screen "83_КалібровкаКрану" 800x454, template "Template_1"
   on GenerateScreen: SetTag("Tag_ScreenNumber", 83)
   IOField "I/O field_3" at 365,32 size 70x25; FormatPattern 99999
      ProcessValue <- "HMI_DB_Calibration_Crane_CurrentStep"
   IOField "I/O field_4" at 365,32 size 70x25; FormatPattern 99999
      ProcessValue <- "HMI_DB_Calibration_Crane_CurrentStep"
      Visibility <- "HMI_DB_Calibration_Crane_Calibrated"
   IOField "I/O field_5" at 365,32 size 70x25; FormatPattern 99999
      ProcessValue <- "HMI_DB_Calibration_Crane_CurrentStep"
      Visibility <- "HMI_DB_Calibration_Crane_Active"
   IOField "I/O field_6" at 365,32 size 70x25; FormatPattern 99999
      ProcessValue <- "HMI_DB_Calibration_Crane_CurrentStep"
      Visibility <- "HMI_DB_Calibration_Crane_Aborted"
   IOField "I/O field_7" at 365,32 size 70x25; FormatPattern 99999
      ProcessValue <- "HMI_DB_Calibration_Crane_CurrentStep"
      Visibility <- "HMI_DB_Calibration_Crane_Fault"
   TextField "Text field_12" at 681,263 size 30x18; Text '110'
   TextField "Text field_13" at 23,263 size 22x18; Text '10'
   TextField "Text field_14" at 89,263 size 22x18; Text '20'
   TextField "Text field_15" at 155,263 size 22x18; Text '30'
   TextField "Text field_16" at 221,263 size 22x18; Text '40'
   TextField "Text field_17" at 288,263 size 22x18; Text '50'
   TextField "Text field_18" at 354,263 size 22x18; Text '60'
   TextField "Text field_19" at 420,263 size 22x18; Text '70'
   TextField "Text field_20" at 486,263 size 22x18; Text '80'
   TextField "Text field_21" at 553,263 size 22x18; Text '90'
   TextField "Text field_22" at 615,263 size 30x18; Text '100'
   TextField "Text field_24" at 748,263 size 30x18; Text '130'
   TextField "Text field_5" at 8,101 size 61x18; Text 'Позиція'
   TextField "Text field_6" at 8,166 size 136x18; Text 'Реперний вимикач'
   TextField "Text field_7" at 8,121 size 80x18; Text 'Швидкість'
   TextField "Text field_8" at 365,142 size 104x18; Text 'Залишок часу'
   IOField "I/O field_1" at 136,98 size 120x25; FormatPattern s999999
      ProcessValue <- "HMI_DB_Calibration_Crane_Position4BR1_mm"
   IOField "I/O field_2" at 136,118 size 120x25; FormatPattern s9999.99
      ProcessValue <- "HMI_DB_Calibration_Crane_Drive1Velocity_rpm"
   Circle "Circle_49" at 211,167 size 16x16
      Appearance <- "HMI_DB_Calibration_Crane_Reference4K1"
   TextField "Text field_9" at 47,5 size 247x21; Text 'Статус калібровки мех. крану'
   TextField "Text field_10" at 482,5 size 181x21; Text 'Поточний крок та дія'
   Group "Group_1" at 365,32 size 70x25
   SymbolicIOField "Symbolic I/O field_1" at 453,29 size 327x32; TextOff '0'; TextOn '1'; TextList "CraneStepName"
      ProcessValue <- "HMI_DB_Calibration_Crane_CurrentStep"
   TextField "Text field_11" at 365,102 size 268x18; Text 'Умови переходу на наступний крок:'
   SymbolicIOField "Symbolic I/O field_2" at 365,115 size 416x32; TextOff '0'; TextOn '1'; TextList "CraneCondition"
      ProcessValue <- "HMI_DB_Calibration_Crane_CurrentStep"
   Group "Group_2" at 680,256 size 32x32
   Group "Group_3" at 18,256 size 32x32
   Group "Group_4" at 84,256 size 32x32
   Group "Group_5" at 150,256 size 32x32
   Group "Group_6" at 216,256 size 32x32
   Group "Group_7" at 283,256 size 32x32
   Group "Group_8" at 349,256 size 32x32
   Group "Group_9" at 415,256 size 32x32
   Group "Group_10" at 481,256 size 32x32
   Group "Group_11" at 548,256 size 32x32
   Group "Group_12" at 614,256 size 32x32
   Group "Group_14" at 747,256 size 32x32
   TextField "Text field_23" at 0,295 size 68x28; Text 'Перевірка умов'
   TextField "Text field_25" at 68,295 size 65x40; Text 'Натисніть кнопку "Вліво"'
   TextField "Text field_26" at 133,295 size 67x40; Text 'Рух до реперної точки 4К1'
   TextField "Text field_27" at 198,295 size 69x40; Text 'Відпустіть кнопку "Вліво"'
   TextField "Text field_28" at 263,295 size 85x40; Text 'Перемістить механізм від 4К1'
   TextField "Text field_29" at 330,295 size 70x28; Text 'Відхід завершено'
   TextField "Text field_30" at 399,295 size 65x40; Text 'Натисніть кнопку "Вліво"'
   TextField "Text field_31" at 462,295 size 70x40; Text 'Повторний підхід до 4К1'
   TextField "Text field_32" at 544,295 size 40x28; Text 'Quick Stop'
   TextField "Text field_33" at 593,295 size 75x40; Text 'Очікування зупинки приводів'
   TextField "Text field_34" at 665,295 size 66x40; Text 'Запуск preset енкодерів'
   TextField "Text field_35" at 725,295 size 75x40; Text 'Калібровку успішно завершено'
   Group "Group_13" at 26,342 size 16x16
   Group "Group_15" at 92,342 size 16x16
   Group "Group_16" at 158,342 size 16x16
   Group "Group_17" at 224,342 size 16x16
   Group "Group_18" at 291,342 size 16x16
   Group "Group_19" at 357,342 size 16x16
   Group "Group_20" at 423,342 size 16x16
   Group "Group_21" at 489,342 size 16x16
   Group "Group_22" at 556,342 size 16x16
   Group "Group_23" at 622,342 size 16x16
   Group "Group_24" at 688,342 size 16x16
   Group "Group_25" at 755,342 size 16x16
   TextField "Text field_36" at 18,381 size 148x18; Text 'Умовні позначення:'
   TextField "Text field_37" at 190,381 size 85x18; Text '- Виконано'
   TextField "Text field_38" at 365,381 size 124x18; Text '- Поточний крок'
   TextField "Text field_39" at 540,381 size 92x18; Text '- Очікується'
   TextField "Text field_40" at 218,226 size 367x21; Text 'Послідовність кроків калібровки мех. крану'
   IOField "I/O field_8" at 540,139 size 60x25; FormatPattern 999; Unit  хв :
      ProcessValue <- "HMI_DB_Calibration_Crane_TimerRemaining_Min"
   IOField "I/O field_9" at 594,139 size 55x25; FormatPattern 999; Unit  сек
      ProcessValue <- "HMI_DB_Calibration_Crane_TimerRemaining_Sec"
   TextField "Text field_42" at 8,141 size 88x18; Text 'Інкременти'
   IOField "I/O field_10" at 136,138 size 80x25; FormatPattern s99999999
      ProcessValue <- "RawPosition"
   Group "Group" at 38,33 size 258x23
   TextField "Text field_43" at 8,191 size 220x18; Text 'Дозв. від мех. підйому і візка'
   Circle "Circle_53" at 211,192 size 16x16
      Appearance <- "HMI_DB_Calibration_Crane_PrerequisitesNotOK"
   IOField "I/O field_11" at 224,98 size 120x25; FormatPattern s999999; Unit  мм
      ProcessValue <- "HMI_DB_Calibration_Crane_Position4BR2_mm"
   IOField "I/O field_12" at 224,118 size 120x25; FormatPattern s9999.99; Unit  об/хв
      ProcessValue <- "HMI_DB_Calibration_Crane_Drive2Velocity_rpm"
   IOField "I/O field_13" at 227,138 size 80x25; FormatPattern s99999999
      ProcessValue <- "RawPosition"
   Circle "Circle_14" at 26,342 size 16x16
      Visibility <- "HMI_DB_Calibration_Crane_Steps_Active_Step10"
   Circle "Circle_15" at 26,342 size 16x16
      Visibility <- "HMI_DB_Calibration_Crane_Steps_Completed_Step10"
   Circle "Circle_17" at 92,342 size 16x16
      Visibility <- "HMI_DB_Calibration_Crane_Steps_Active_Step20"
   Circle "Circle_18" at 92,342 size 16x16
      Visibility <- "HMI_DB_Calibration_Crane_Steps_Completed_Step20"
   Circle "Circle_20" at 158,342 size 16x16
      Visibility <- "HMI_DB_Calibration_Crane_Steps_Active_Step30"
   Circle "Circle_21" at 158,342 size 16x16
      Visibility <- "HMI_DB_Calibration_Crane_Steps_Completed_Step30"
   Circle "Circle_23" at 224,342 size 16x16
      Visibility <- "HMI_DB_Calibration_Crane_Steps_Active_Step40"
   Circle "Circle_24" at 224,342 size 16x16
      Visibility <- "HMI_DB_Calibration_Crane_Steps_Completed_Step40"
   Circle "Circle_26" at 291,342 size 16x16
      Visibility <- "HMI_DB_Calibration_Crane_Steps_Active_Step50"
   Circle "Circle_27" at 291,342 size 16x16
      Visibility <- "HMI_DB_Calibration_Crane_Steps_Completed_Step50"
   Circle "Circle_29" at 357,342 size 16x16
      Visibility <- "HMI_DB_Calibration_Crane_Steps_Active_Step60"
   Circle "Circle_30" at 357,342 size 16x16
      Visibility <- "HMI_DB_Calibration_Crane_Steps_Completed_Step60"
   Circle "Circle_32" at 423,342 size 16x16
      Visibility <- "HMI_DB_Calibration_Crane_Steps_Active_Step70"
   Circle "Circle_33" at 423,342 size 16x16
      Visibility <- "HMI_DB_Calibration_Crane_Steps_Completed_Step70"
   Circle "Circle_35" at 489,342 size 16x16
      Visibility <- "HMI_DB_Calibration_Crane_Steps_Active_Step80"
   Circle "Circle_36" at 489,342 size 16x16
      Visibility <- "HMI_DB_Calibration_Crane_Steps_Completed_Step80"
   Circle "Circle_38" at 556,342 size 16x16
      Visibility <- "HMI_DB_Calibration_Crane_Steps_Active_Step90"
   Circle "Circle_39" at 556,342 size 16x16
      Visibility <- "HMI_DB_Calibration_Crane_Steps_Completed_Step90"
   Circle "Circle_41" at 622,342 size 16x16
      Visibility <- "HMI_DB_Calibration_Crane_Steps_Active_Step100"
   Circle "Circle_42" at 622,342 size 16x16
      Visibility <- "HMI_DB_Calibration_Crane_Steps_Completed_Step100"
   Circle "Circle_44" at 688,342 size 16x16
      Visibility <- "HMI_DB_Calibration_Crane_Steps_Active_Step110"
   Circle "Circle_45" at 688,342 size 16x16
      Visibility <- "HMI_DB_Calibration_Crane_Steps_Completed_Step110"
   Circle "Circle_47" at 755,342 size 16x16
      Visibility <- "HMI_DB_Calibration_Crane_Steps_Active_Step130"
   Circle "Circle_48" at 755,342 size 16x16
      Visibility <- "HMI_DB_Calibration_Crane_Steps_Completed_Step130"
   TextField "Text field_41" at 83,33 size 169x23; Text 'НЕ КАЛІБРОВАНО'
      Visibility <- "HMI_DB_Calibration_Crane_Calibrated"
   TextField "Text field_4" at 38,33 size 258x23; Text 'КАЛІБРОВКА АНУЛЬОВАНА'
      Visibility <- "HMI_DB_Calibration_Crane_Aborted"
   TextField "Text field_2" at 58,33 size 219x23; Text 'КАЛІБРОВКА АКТИВНА'
      Visibility <- "HMI_DB_Calibration_Crane_Active"
   TextField "Text field_3" at 56,33 size 223x23; Text 'ПОМИЛКА КАЛІБРОВКИ'
      Visibility <- "HMI_DB_Calibration_Crane_Fault"
   TextField "Text field_1" at 98,33 size 139x23; Text 'КАЛІБРОВАНО'
      Visibility <- "HMI_DB_Calibration_Crane_Calibrated"
   TextField "Text field_44" at 149,77 size 75x18; Text '4М1'
   TextField "Text field_45" at 221,77 size 75x18; Text '4М2'
   Group "Group_26" at 207,61 size 25x0
   Line "Line_4" at 207,61 size 25x0
      Visibility <- "HMI_DB_Crane_movement_mechanism_FirstSpeedRight"
   Line "Line_5" at 207,61 size 25x0
      Visibility <- "HMI_DB_Crane_movement_mechanism_FirstSpeedLeft"

screen "70_Діагностика" 800x454, template "Template_1"
   on GenerateScreen: SetTag("Tag_ScreenNumber", 70); function_c655a98f("HMI_Connection_1", "HMI_PLC_Mode"); "HMI_UpdateCommunication"()
   TextField "Text field_1" at 166,42 size 46x23; Text 'A1.1'
   TextField "Text field_2" at 166,216 size 46x23; Text 'A1.0'
   TextField "Text field_3" at 715,26 size 41x23; Text '1BR'
   TextField "Text field_4" at 715,115 size 41x23; Text '3BR'
   TextField "Text field_5" at 710,206 size 52x23; Text '4BR1'
   TextField "Text field_6" at 710,295 size 52x23; Text '4BR2'
   TextField "Text field_7" at 436,67 size 46x23; Text 'A1.6'
   TextField "Text field_8" at 348,286 size 23x18; Text 'U1'
   TextField "Text field_9" at 394,286 size 40x18; Text '1UZ1'
   TextField "Text field_10" at 436,286 size 40x18; Text '3UZ1'
   TextField "Text field_11" at 479,286 size 40x18; Text '4UZ1'
   TextField "Text field_12" at 522,286 size 40x18; Text '4UZ2'
   Button "Button_3" at 4,10 size 104x34; TextOff 'Діагностика / Тренди'; TextOn 'Діагностика'
      on Release: ActivateScreen("50_Trends(1UZ1)", 0)
   TextField "PN_Status_DisplayOpen" at 120,1 size 550x20; Text 'MRP: RING OPEN / MRP: КІЛЬЦЕ РОЗІМКНЕНЕ'
      Visibility <- "HMI_Show_RingOpen"
   TextField "PN_Status_DisplayClosed" at 120,0 size 550x20; Text 'MRP: RING CLOSED / MRP: КІЛЬЦЕ ЗАМКНЕНЕ'
      Visibility <- "HMI_Show_RingClosed"
   TextField "PN_Status_DisplayUnknown" at 120,20 size 550x20; Text 'PN: DIAGNOSTIC DATA UNAVAILABLE / PN: ДІАГНОСТИЧНІ ДАНІ НЕДОСТУПНІ'
      Visibility <- "HMI_Show_DiagnosticsUnknown"
   TextField "PN_Status_DisplayHmiFault" at 120,20 size 550x20; Text 'HMI: PLC DETECTED A PANEL COMMUNICATION FAULT / HMI: ПЛК ВИЯВИВ ПОРУШЕННЯ ОБМІНУ З ПАНЕЛЛЮ'
      Visibility <- "HMI_Show_PanelFault"
   TextField "HMI_Status_NoConnection" at 120,20 size 550x20; Text 'HMI: NO COMMUNICATION BETWEEN PLC AND OPERATOR PANEL / HMI: НЕМАЄ ЗВʼЯЗКУ МІЖ ПЛК І ПАНЕЛЛЮ ОПЕРАТОРА'
      Visibility <- "HMI_Show_NoConnection"
   TextField "HMI_Status_CpuStopped" at 120,20 size 550x20; Text 'PLC: STOPPED. DIAGNOSTICS ARE NOT UPDATING / ПЛК: ЗУПИНЕНО (STOP). ДІАГНОСТИКА НЕ ОНОВЛЮЄТЬСЯ'
      Visibility <- "HMI_Show_CpuStopped"
   TextField "HMI_Status_CpuUnknown" at 120,20 size 550x20; Text 'PLC: RUN MODE NOT CONFIRMED / ПЛК: РЕЖИМ RUN НЕ ПІДТВЕРДЖЕНО'
      Visibility <- "HMI_Show_CpuUnknown"
   GraphicView "Graphic view_1" at 64,63 size 255x119; Picture "plc"
   GraphicView "Graphic view_2" at 428,91 size 62x124; Picture "scalance"
   GraphicView "Graphic view_3" at 697,30 size 76x48; Picture "6FX2001-5QN25_P_NC01_XX_01618I"
   GraphicView "Graphic view_5" at 343,307 size 46x80; Picture "6SL3040-1MA01-0AA0_P_D211_XX_00205P"
   GraphicView "Graphic view_6" at 697,119 size 76x48; Picture "6FX2001-5QN25_P_NC01_XX_01618I"
   GraphicView "Graphic view_7" at 697,209 size 76x48; Picture "6FX2001-5QN25_P_NC01_XX_01618I"
   GraphicView "Graphic view_8" at 697,299 size 76x48; Picture "6FX2001-5QN25_P_NC01_XX_01618I"
   GraphicView "Graphic view_4" at 100,239 size 184x118; Picture "hmi_1"
   GraphicView "Graphic view_9" at 389,301 size 50x90; Picture "6SL3210-1PE14-3UL1_P_D011_XX_00576_4_1"
   GraphicView "Graphic view_10" at 431,301 size 50x90; Picture "6SL3210-1PE14-3UL1_P_D011_XX_00576_4_1"
   GraphicView "Graphic view_11" at 474,301 size 50x90; Picture "6SL3210-1PE14-3UL1_P_D011_XX_00576_4_1"
   GraphicView "Graphic view_12" at 517,301 size 50x90; Picture "6SL3210-1PE14-3UL1_P_D011_XX_00576_4_1"
   Group "NOK_A1.5" at 276,66 size 40x111
   Group "NOK_A1.4" at 233,66 size 40x111
   Group "NOK_A1.3" at 192,66 size 40x111
   Group "NOK_A1.2" at 147,66 size 40x111
   Group "NOK_A1.1" at 66,66 size 77x111
   GraphicView "Graphic view_21" at 343,309 size 45x80; Picture "Graphic_4"
      Visibility <- "HMI_DB_Alarms_Diagn_AlarmWord1"
   GraphicView "Graphic view_20" at 391,309 size 45x80; Picture "Graphic_4"
      Visibility <- "HMI_DB_Alarms_Diagn_AlarmWord1"
   GraphicView "Graphic view_19" at 431,309 size 45x80; Picture "Graphic_4"
      Visibility <- "HMI_DB_Alarms_Diagn_AlarmWord1"
   GraphicView "Graphic view_18" at 479,309 size 45x80; Picture "Graphic_4"
      Visibility <- "HMI_DB_Alarms_Diagn_AlarmWord1"
   GraphicView "Graphic view_17" at 519,309 size 45x80; Picture "Graphic_4"
      Visibility <- "HMI_DB_Alarms_Diagn_AlarmWord1"
   GraphicView "Graphic view_16" at 688,290 size 85x80; Picture "Graphic_4"
      Visibility <- "HMI_DB_Alarms_Diagn_AlarmWord1"
   GraphicView "Graphic view_15" at 688,202 size 85x80; Picture "Graphic_4"
      Visibility <- "HMI_DB_Alarms_Diagn_AlarmWord1"
   GraphicView "Graphic view_14" at 688,114 size 85x80; Picture "Graphic_4"
      Visibility <- "HMI_DB_Alarms_Diagn_AlarmWord1"
   GraphicView "Graphic view_13" at 688,26 size 85x80; Picture "Graphic_4"
      Visibility <- "HMI_DB_Alarms_Diagn_AlarmWord1"
   GraphicView "Graphic view_22" at 416,96 size 85x106; Picture "Graphic_4"
      Visibility <- "HMI_DB_Alarms_Diagn_AlarmWord1"
   GraphicView "Graphic view_23" at 279,348 size 40x70; Picture "Graphic_4"
      Visibility <- "HMI_Show_Cross_HMI_CU"
   GraphicView "Graphic view_24" at 287,172 size 40x70; Picture "Graphic_4"
      Visibility <- "HMI_Show_Cross_PLC_SC"
   GraphicView "Graphic view_25" at 112,348 size 40x70; Picture "Graphic_4"
      Visibility <- "HMI_Show_Cross_PLC_HMI"
   GraphicView "Graphic view_26" at 383,204 size 40x70; Picture "Graphic_4"
      Visibility <- "HMI_Show_Cross_SC_CU"
   Line "Line_8" at 276,66 size 40x111
      Visibility <- "HMI_DB_Alarms_Diagn_AlarmWord1"
   Line "Line_9" at 276,66 size 40x111
      Visibility <- "HMI_DB_Alarms_Diagn_AlarmWord1"
   Line "Line_1" at 233,66 size 40x111
      Visibility <- "HMI_DB_Alarms_Diagn_AlarmWord1"
   Line "Line_2" at 233,66 size 40x111
      Visibility <- "HMI_DB_Alarms_Diagn_AlarmWord1"
   Line "Line_3" at 192,66 size 40x111
      Visibility <- "HMI_DB_Alarms_Diagn_AlarmWord1"
   Line "Line_4" at 192,66 size 40x111
      Visibility <- "HMI_DB_Alarms_Diagn_AlarmWord1"
   Line "Line_5" at 147,66 size 40x111
      Visibility <- "HMI_DB_Alarms_Diagn_AlarmWord1"
   Line "Line_6" at 147,66 size 40x111
      Visibility <- "HMI_DB_Alarms_Diagn_AlarmWord1"
   Line "Line_7" at 66,66 size 77x111
      Visibility <- "HMI_DB_Alarms_Diagn_AlarmWord1"
   Line "Line_10" at 66,66 size 77x111
      Visibility <- "HMI_DB_Alarms_Diagn_AlarmWord1"
   Button "btn1BR" at 690,32 size 90x45; TextOff 'Text'
      on Release: ActivateScreen("77_1BR", 0)
   Button "btn3BR" at 690,121 size 90x45; TextOff 'Text'
      on Release: ActivateScreen("78_3BR", 0)
   Button "btn4BR1" at 690,211 size 90x45; TextOff 'Text'
      on Release: ActivateScreen("79_4BR1", 0)
   Button "btn4BR2" at 690,301 size 90x45; TextOff 'Text'
      on Release: ActivateScreen("710_4BR2", 0)
   Button "btnU1" at 330,304 size 62x92; TextOff 'Text'
      on Release: ActivateScreen("30_Drives(CU)", 0)
   Button "btnA1.2" at 147,50 size 43x119; TextOff 'Text'
      on Release: ActivateScreen("71_A1.2(DI32)_1", 0)
   Button "btnA1.3" at 189,50 size 43x119; TextOff 'Text'
      on Release: ActivateScreen("73_A1.3(DI32)_1", 0)
   Button "btnA1.4" at 233,50 size 43x119; TextOff 'Text'
      on Release: ActivateScreen("76_A1.4(IW8)", 0)
   Button "btnA1.5" at 276,50 size 43x119; TextOff 'Text'
      on Release: ActivateScreen("75_A1.5(DQ16)", 0)
   Button "btn1UZ1" at 394,304 size 35x92; TextOff 'Text'
      on Release: ActivateScreen("31_Drives(1UZ1)", 0)
   Button "btn3UZ1" at 434,304 size 37x92; TextOff 'Text'
      on Release: ActivateScreen("32_Drives(3UZ1)", 0)
   Button "btn4UZ1" at 478,304 size 37x92; TextOff 'Text'
      on Release: ActivateScreen("33_Drives(4UZ1)", 0)
   Button "btn4UZ2" at 522,304 size 37x92; TextOff 'Text'
      on Release: ActivateScreen("34_Drives(4UZ2)", 0)

VB script "StartLog"
   'Tip:
   ' 1. Use the <CTRL+SPACE> or <CTRL+I> shortcut to open a list of all objects and functions
   ' 2. Write the code using the HMI Runtime object.
   '  Example: HmiRuntime.Screens("Screen_1").
   ' 3. Use the <CTRL+J> shortcut to create an object reference.
   'Write the code as of this position:
    bb0abc73-aec8-40d0-9880-0280a6a3de42()
    fd9437ed-c09f-45a2-bbcf-d542009dcc27 $3$hmiDataLog$,1UZ1
    fd9437ed-c09f-45a2-bbcf-d542009dcc27 $3$hmiDataLog$, 3UZ1 
    fd9437ed-c09f-45a2-bbcf-d542009dcc27 $3$hmiDataLog$, 4UZ1 
    fd9437ed-c09f-45a2-bbcf-d542009dcc27 $3$hmiDataLog$,4UZ2 
    fd9437ed-c09f-45a2-bbcf-d542009dcc27 $3$hmiAlarmLog$,MessageContactor 
    fd9437ed-c09f-45a2-bbcf-d542009dcc27 $3$hmiAlarmLog$,MessageLiftUp 
    fd9437ed-c09f-45a2-bbcf-d542009dcc27 $3$hmiAlarmLog$,MessageTrolley 
    fd9437ed-c09f-45a2-bbcf-d542009dcc27 $3$hmiAlarmLog$,MessageCrane 
    fd9437ed-c09f-45a2-bbcf-d542009dcc27 $3$hmiAlarmLog$,MessageDiag 
    fd9437ed-c09f-45a2-bbcf-d542009dcc27 $3$hmiAlarmLog$,AlarmCrane 
    fd9437ed-c09f-45a2-bbcf-d542009dcc27 $3$hmiAlarmLog$,AlarmTrolley 
    fd9437ed-c09f-45a2-bbcf-d542009dcc27 $3$hmiAlarmLog$,AlarmLiftUp 
    fd9437ed-c09f-45a2-bbcf-d542009dcc27 $3$hmiAlarmLog$,AlarmContactor 
    fd9437ed-c09f-45a2-bbcf-d542009dcc27 $3$hmiAlarmLog$,AlarmDiag 
    fd9437ed-c09f-45a2-bbcf-d542009dcc27 $3$hmiAlarmLog$,MessageSelf 
    SmartTags("iStep") = 0

VB script "StopLog"
   'Tip:
   ' 1. Use the <CTRL+SPACE> or <CTRL+I> shortcut to open a list of all objects and functions
   ' 2. Write the code using the HMI Runtime object.
   '  Example: HmiRuntime.Screens "Screen_1" .
   ' 3. Use the <CTRL+J> shortcut to create an object reference.
   'Write the code as of this position:
    b6526003-1e6c-4105-b1c3-8571bad56740 $3$hmiDataLog$,1UZ1
    b6526003-1e6c-4105-b1c3-8571bad56740 $3$hmiDataLog$,3UZ1 
    b6526003-1e6c-4105-b1c3-8571bad56740 $3$hmiDataLog$,4UZ1 
    b6526003-1e6c-4105-b1c3-8571bad56740 $3$hmiDataLog$,4UZ2 
    b6526003-1e6c-4105-b1c3-8571bad56740 $3$hmiAlarmLog$,MessageContactor 
    b6526003-1e6c-4105-b1c3-8571bad56740 $3$hmiAlarmLog$,MessageLiftUp 
    b6526003-1e6c-4105-b1c3-8571bad56740 $3$hmiAlarmLog$,MessageTrolley 
    b6526003-1e6c-4105-b1c3-8571bad56740 $3$hmiAlarmLog$,MessageCrane 
    b6526003-1e6c-4105-b1c3-8571bad56740 $3$hmiAlarmLog$,MessageDiag 
    b6526003-1e6c-4105-b1c3-8571bad56740 $3$hmiAlarmLog$,AlarmCrane 
    b6526003-1e6c-4105-b1c3-8571bad56740 $3$hmiAlarmLog$,AlarmTrolley 
    b6526003-1e6c-4105-b1c3-8571bad56740 $3$hmiAlarmLog$,AlarmLiftUp 
    b6526003-1e6c-4105-b1c3-8571bad56740 $3$hmiAlarmLog$,AlarmContactor 
    b6526003-1e6c-4105-b1c3-8571bad56740 $3$hmiAlarmLog$,AlarmDiag 
    b6526003-1e6c-4105-b1c3-8571bad56740 $3$hmiAlarmLog$,MessageSelf 
    efd5fb8c-e901-419b-bc1e-08a47a763dd7  
    SmartTags("iStep")  = 1

VB script "CopyLogs"
   'Tip:
   ' 1. Use the <CTRL+SPACE> or <CTRL+I> shortcut to open a list of all objects and functions
   ' 2. Write the code using the HMI Runtime object.
   '  Example: HmiRuntime.Screens("Screen_1").
   ' 3. Use the <CTRL+J> shortcut to create an object reference.
   'Write the code as of this position:
    
    Dim st
    
    On Error Resume Next
    
    e9be9208-412d-4969-b0d9-b24c90392a10 $3$hmiDataLog$,1UZ1, "\Storage Card USB\archive\", $3$hmiCopy$
    e9be9208-412d-4969-b0d9-b24c90392a10 $3$hmiDataLog$,3UZ1, "\Storage Card USB\archive\", $3$hmiCopy$
    e9be9208-412d-4969-b0d9-b24c90392a10 $3$hmiDataLog$,4UZ1, "\Storage Card USB\archive\", $3$hmiCopy$
    e9be9208-412d-4969-b0d9-b24c90392a10 $3$hmiDataLog$,4UZ2, "\Storage Card USB\archive\", $3$hmiCopy$
    e9be9208-412d-4969-b0d9-b24c90392a10 $3$hmiAlarmLog$,MessageContactor,  "\Storage Card USB\archive\", $3$hmiCopy$
    e9be9208-412d-4969-b0d9-b24c90392a10 $3$hmiAlarmLog$,MessageLiftUp, "\Storage Card USB\archive\", $3$hmiCopy$
    e9be9208-412d-4969-b0d9-b24c90392a10 $3$hmiAlarmLog$,MessageTrolley, "\Storage Card USB\archive\", $3$hmiCopy$
    e9be9208-412d-4969-b0d9-b24c90392a10 $3$hmiAlarmLog$,MessageCrane,  "\Storage Card USB\archive\", $3$hmiCopy$
    e9be9208-412d-4969-b0d9-b24c90392a10 $3$hmiAlarmLog$,MessageDiag,  "\Storage Card USB\archive\", $3$hmiCopy$
    e9be9208-412d-4969-b0d9-b24c90392a10 $3$hmiAlarmLog$,AlarmCrane,  "\Storage Card USB\archive\", $3$hmiCopy$
    e9be9208-412d-4969-b0d9-b24c90392a10 $3$hmiAlarmLog$,AlarmTrolley,  "\Storage Card USB\archive\", $3$hmiCopy$
    e9be9208-412d-4969-b0d9-b24c90392a10 $3$hmiAlarmLog$,AlarmLiftUp,  "\Storage Card USB\archive\", $3$hmiCopy$
    e9be9208-412d-4969-b0d9-b24c90392a10 $3$hmiAlarmLog$,AlarmContactor,  "\Storage Card USB\archive\", $3$hmiCopy$
    e9be9208-412d-4969-b0d9-b24c90392a10 $3$hmiAlarmLog$,AlarmDiag,  "\Storage Card USB\archive\", $3$hmiCopy$
    e9be9208-412d-4969-b0d9-b24c90392a10 $3$hmiAlarmLog$,MessageSelf,  "\Storage Card USB\archive\", $3$hmiCopy$
    SmartTags("iStep") = 2
    

VB script "HMI_UpdateCommunication"
   ' Стан з’єднання визначають системні повідомлення самої панелі.
   ' 140001 (розрив): HMI_Show_NoConnection = 1; 140000 (відновлення): = 0.
   ' Це внутрішній тег HMI: його значення не залежить від доступності ПЛК.
   ' Скрипт не перезаписує цей тег прочитаними з кешу даними.
   Dim connected, mode, running, panelFault, diagUnknown, item
   connected = Not CBool(SmartTags("HMI_Show_NoConnection"))
   mode = CInt(SmartTags("HMI_PLC_Mode"))
   If Not connected Then
       ' Скидаємо останній режим, щоб після відновлення дочекатися нового GetPLCMode.
       If mode <> 0 Then SmartTags("HMI_PLC_Mode") = 0
       mode = 0
   End If
   running = connected And (mode = 8)
   SmartTags("HMI_Show_CpuStopped") = connected And (mode = 4)
   SmartTags("HMI_Show_CpuUnknown") = connected And (mode <> 4) And (mode <> 8)
   
   If running Then
       ' Назва старого HMI-тега містить Fault, але він читає DisplayHmiNoFault.
       panelFault = Not CBool(SmartTags("PN_Diagnostics_DisplayHmiFault"))
       diagUnknown = CBool(SmartTags("PN_Diagnostics_DisplayUnknown"))
       SmartTags("HMI_Show_PanelFault") = panelFault
       SmartTags("HMI_Show_DiagnosticsUnknown") = diagUnknown And Not panelFault
       SmartTags("HMI_Show_RingOpen") = CBool(SmartTags("PN_Diagnostics_DisplayOpen"))
       SmartTags("HMI_Show_RingClosed") = CBool(SmartTags("PN_Diagnostics_DisplayClosed"))
       SmartTags("HMI_Show_Cross_PLC_HMI") = CBool(SmartTags("HMI_DB_Diagnostics_Ring_PLC_HMI_NOK"))
       SmartTags("HMI_Show_Cross_PLC_SC") = CBool(SmartTags("HMI_DB_Diagnostics_Ring_PLC_SCALAMCE_NOK"))
       SmartTags("HMI_Show_Cross_SC_CU") = CBool(SmartTags("HMI_DB_Diagnostics_Ring_SCALAMCE_CU_NOK"))
       SmartTags("HMI_Show_Cross_HMI_CU") = CBool(SmartTags("HMI_DB_Diagnostics_Ring_HMI_CU_NOK"))
   Else
       ' У STOP або без зв’язку не читаємо зовнішні теги та прибираємо застарілі покази.
       For Each item In Array("PanelFault", "DiagnosticsUnknown", "RingOpen", "RingClosed", "Cross_PLC_HMI", "Cross_PLC_SC", "Cross_SC_CU", "Cross_HMI_CU")
           SmartTags("HMI_Show_" & item) = False
       Next
   End If
*)

(* ===== HMI "HMI_RT_1" =====

ScreenModuleEditorView "fcptAI" 640x480
   IOField "iofData" at 49,12 size 400x18; FormatPattern ???????????????????????????????????????????????
      ProcessValue <- "Data.Text"
   IOField "iofAdress" at 5,12 size 50x18; FormatPattern ?????
      ProcessValue <- "Data.Chanal"
   IOField "iofAdress_1" at 515,12 size 70x18; FormatPattern 99.99; Unit V
      ProcessValue <- "Data.PhyVal"
*)

(* ===== HMI "HMI_RT_1" =====

ScreenModuleEditorView "fcptDI" 640x480
   Circle "crcSignalStatus" at 5,13 size 16x16
      Appearance <- "Data.Val"
   IOField "iofData" at 65,12 size 470x18; FormatPattern ????????????????????????????????????????????????????????
      ProcessValue <- "Data.Text"
   IOField "iofAdress" at 21,12 size 50x18; FormatPattern ?????
      ProcessValue <- "Data.Chanal"
*)

(* ===== HMI "HMI_RT_1" =====

ScreenModuleEditorView "fcptDO" 640x480
   Circle "crcSignalStatus" at 5,13 size 16x16
      Appearance <- "Data.Val"
   IOField "iofData" at 65,12 size 470x18; FormatPattern ????????????????????????????????????????????????????????
      ProcessValue <- "Data.Text"
   IOField "iofAdress" at 21,12 size 50x18; FormatPattern ?????
      ProcessValue <- "Data.Chanal"
*)